Staubli VAL3: sensorFilter.pgx

public program sensorFilter(num& x_nFTData[], num& x_nFTValue[])
  local num l_nNum
  local num l_n
  local num l_nFTTemp
  local num l_nWight[40]
  local num l_nTemp
  local num l_i
  local num l_j
  local num l_nFTData[40]
begin

  //This program is used for filtering the noise of the F/T sensor itself, Thus the robot can
  //move smoothly. And the filter algrithm can be replaced when you need.


  //Moving Average Filter
  l_nNum=4
  l_nFTTemp=0
  for l_n=0 to l_nNum-1
    l_nFTTemp=l_nFTTemp+x_nFTData[l_n]
  endFor
  x_nFTValue=l_nFTTemp/l_nNum

  //Weighted Recursive Average Filter
  l_nNum=4
  l_nFTTemp=0
  l_nWight[0]=0.5
  l_nWight[1]=0.3413
  l_nWight[2]=0.1359
  l_nWight[3]=0.0215
  l_nWight[4]=0.0013
  for l_n=0 to l_nNum
    l_nFTTemp=l_nFTTemp+x_nFTData[l_n]*l_nWight[l_n]
  endFor
  x_nFTValue=l_nFTTemp

  //Median Average Filter
  l_nFTTemp=0
  l_nNum=4
  l_nFTData=x_nFTData

  for l_j=0 to l_nNum-1
    for l_i=0 to l_nNum-1-l_j
      if l_nFTData[l_i]>l_nFTData[l_i+1]
        l_nFTData=l_nFTData[l_i]
        l_nFTData[l_i]=l_nFTData[l_i+1]
        l_nFTData[l_i+1]=l_nTemp
      endIf
    endFor
  endFor

  for l_i=1 to l_nNum-1
    l_nFTTemp=l_nFTTemp+l_nFTData[l_i]
  endFor

  x_nFTValue=l_nFTTemp/(l_nNum-2)

  //Lowpass Filter



  //Kalman Filter



end
